// TIA Portal V17 export
// export: Created 2023-09-11T21:11:16.7675034Z, ExportSetting WithDefaults, DisplayName Totally Integrated Automation Portal, DisplayVersion V17 Update 6, DisplayName TIA Portal Openness, DisplayVersion V17 Update 6, DisplayName TIA Portal Teamcenter Gateway, DisplayVersion V17 Update 6, DisplayName TIA Portal Version Control Interface, DisplayVersion V17, DisplayName Simotion SCOUT TIA, DisplayVersion 5.4.3.0, DisplayName TIA Portal Test Suite Advanced, DisplayVersion V17 Update 1, DisplayName SIMOCODE ES, DisplayVersion V17 Update 5, DisplayName SINAMICS Startdrive Advanced, DisplayVersion V17 SP1, DisplayName SINAMICS Startdrive G130, G150, S120, S150, SINAMICS MV, S210, DisplayVersion V17 SP1, DisplayName SINAMICS Startdrive G110M, G120, G120C, G120D, G120P, G115D, DisplayVersion V17 SP1, DisplayName SIRIUS Safety ES, DisplayVersion V17 Update 5, DisplayName STEP 7 Professional, DisplayVersion V17 Update 6, DisplayName STEP 7 CFC, DisplayVersion V17 Update 1, DisplayName STEP 7 Safety, DisplayVersion V17 Update 6, DisplayName WinCC Advanced, DisplayVersion V17 Update 6, DisplayName SIMATIC Visualization Architect, DisplayVersion V17 Update 5
FUNCTION "08_Gate Manager" : Void   // FC9, F_LAD
{ S7_Optimized_Access := 'TRUE' }
VERSION : 0.1
// stored: AutoNumber true, IsIECCheckEnabled false, UDAEnableTagReadback false
   VAR_TEMP
      temp_EXAMPLE_OPEN : Bool;
   END_VAR
BEGIN

REGION Network 1: !!COLUMN_1$$
   // Sorter Gate
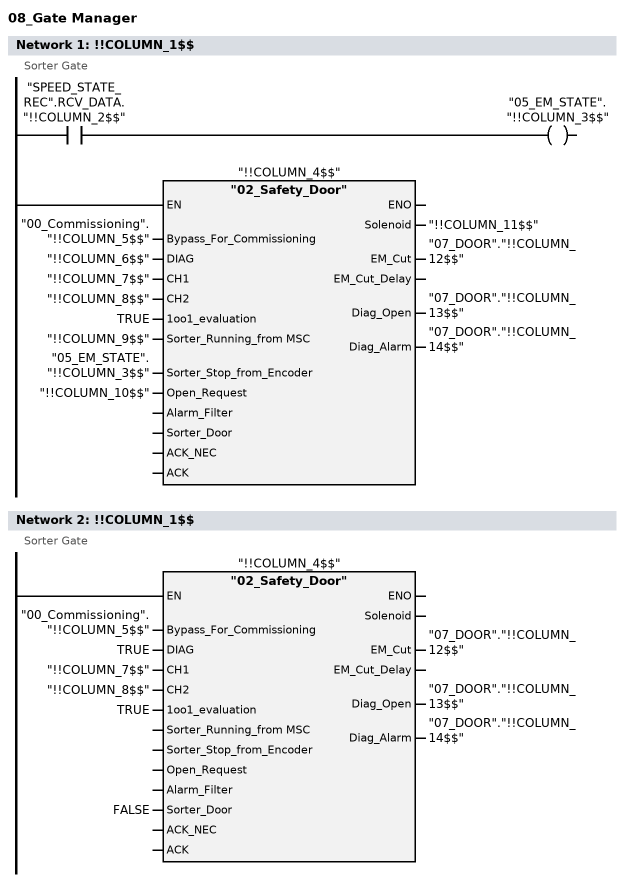
   RUNG wire#powerrail
      Contact( "SPEED_STATE_REC".RCV_DATA."!!COLUMN_2$$" )
      Coil( "05_EM_STATE"."!!COLUMN_3$$" )
   END_RUNG
   RUNG wire#powerrail
      "!!COLUMN_4$$"(Bypass_For_Commissioning := "00_Commissioning"."!!COLUMN_5$$", DIAG := "!!COLUMN_6$$", CH1 := "!!COLUMN_7$$", CH2 := "!!COLUMN_8$$", "1oo1_evaluation" := TRUE, "Sorter_Running_from MSC" := "!!COLUMN_9$$", Sorter_Stop_from_Encoder := "05_EM_STATE"."!!COLUMN_3$$", Open_Request := "!!COLUMN_10$$", Alarm_Filter :=, Sorter_Door :=, ACK_NEC :=, ACK :=, Solenoid => "!!COLUMN_11$$", EM_Cut => "07_DOOR"."!!COLUMN_12$$", EM_Cut_Delay =>, Diag_Open => "07_DOOR"."!!COLUMN_13$$", Diag_Alarm => "07_DOOR"."!!COLUMN_14$$")
   END_RUNG
   // the same network as SCL:
   "05_EM_STATE"."!!COLUMN_3$$" := "SPEED_STATE_REC".RCV_DATA."!!COLUMN_2$$";
   "!!COLUMN_4$$"(Bypass_For_Commissioning := "00_Commissioning"."!!COLUMN_5$$",   // "02_Safety_Door"
                  DIAG := "!!COLUMN_6$$",
                  CH1 := "!!COLUMN_7$$",
                  CH2 := "!!COLUMN_8$$",
                  "1oo1_evaluation" := TRUE,
                  "Sorter_Running_from MSC" := "!!COLUMN_9$$",
                  Sorter_Stop_from_Encoder := "05_EM_STATE"."!!COLUMN_3$$",
                  Open_Request := "!!COLUMN_10$$",
                  Solenoid => "!!COLUMN_11$$",
                  EM_Cut => "07_DOOR"."!!COLUMN_12$$",
                  Diag_Open => "07_DOOR"."!!COLUMN_13$$",
                  Diag_Alarm => "07_DOOR"."!!COLUMN_14$$");
END_REGION

REGION Network 2: !!COLUMN_1$$
   // Sorter Gate
   RUNG wire#powerrail
      "!!COLUMN_4$$"(Bypass_For_Commissioning := "00_Commissioning"."!!COLUMN_5$$", DIAG := TRUE, CH1 := "!!COLUMN_7$$", CH2 := "!!COLUMN_8$$", "1oo1_evaluation" := TRUE, "Sorter_Running_from MSC" :=, Sorter_Stop_from_Encoder :=, Open_Request :=, Alarm_Filter :=, Sorter_Door := FALSE, ACK_NEC :=, ACK :=, Solenoid =>, EM_Cut => "07_DOOR"."!!COLUMN_12$$", EM_Cut_Delay =>, Diag_Open => "07_DOOR"."!!COLUMN_13$$", Diag_Alarm => "07_DOOR"."!!COLUMN_14$$")
   END_RUNG
   // the same network as SCL:
   "!!COLUMN_4$$"(Bypass_For_Commissioning := "00_Commissioning"."!!COLUMN_5$$",   // "02_Safety_Door"
                  DIAG := TRUE,
                  CH1 := "!!COLUMN_7$$",
                  CH2 := "!!COLUMN_8$$",
                  "1oo1_evaluation" := TRUE,
                  Sorter_Door := FALSE,
                  EM_Cut => "07_DOOR"."!!COLUMN_12$$",
                  Diag_Open => "07_DOOR"."!!COLUMN_13$$",
                  Diag_Alarm => "07_DOOR"."!!COLUMN_14$$");
END_REGION
END_FUNCTION
